TYPE ST_HMIParameters :
STRUCT
	
	tCheckAirFlowTime 	: TIME;					//Time in seconds to check air flow
	
	aM1Position : ARRAY [1..3] OF LREAL;		//M1 Motor - Stage Collection Vertical Axis  |1=HomePosition|2=RecoveryPosition|3=DryPosition|
	aM2Position : ARRAY [1..3] OF LREAL;		//M2 Motor - Sample Recovery Vertical Axis   |1=HomePosition|2=Waste|3=Fill Vials|
	aM3Position : ARRAY [1..5] OF LREAL;		//M3 Motor - Sample Recovery Horizontal Axis |1=HomePosition/Waste|2=VialLine1|3=VialLine2|4=VialLine3|5=VialLine4|
	
	//Stage Collection Motor M1 - Vertical
	rM1Velocity			:	LREAL;
	rM1Accleration		:	LREAL;
	rM1Deceleration		:	LREAL;
	
	//Sample Recovey Motor M2 - Vertical
	rM2Velocity			:	LREAL;
	rM2Accleration		:	LREAL;
	rM2Deceleration		:	LREAL;
	
	//Sample Recovey Motor M3 - Horizontal
	rM3Velocity			:	LREAL;
	rM3Accleration		:	LREAL;
	rM3Deceleration		:	LREAL;
	
	

END_STRUCT
END_TYPE

(* stored: Version 1.1.0.1, ProductVersion 3.1.4024.12
   DUT ST_HMIParameters: Id {615fc2f1-fbaf-4f88-aebf-fc5849c356b3} *)
